FUNCTION ArgAsIComponent : Result
VAR_INPUT
	iSource	: I_Component;
END_VAR
VAR_OUTPUT
	iDest	: I_StateManager;
END_VAR

IF iSource = 0 THEN
	ArgAsIComponent := Err.Itf0;
	RETURN;
END_IF

IF __QUERYINTERFACE(iSource, iDest) THEN
	ArgAsIComponent := Ok;
ELSE
	ArgAsIComponent := Err.NoMatch;
END_IF

END_FUNCTION

(* stored: Version 1.1.0.1
   POU ArgAsIComponent: Id {5c29e6e1-73d7-4b4a-82c7-dcd0d4c36bbf}, SpecialFunc None *)
